FUNCTION_BLOCK FB_NormalWash IMPLEMENTS I_WashStrategy
VAR_INPUT
END_VAR
VAR_OUTPUT
END_VAR
VAR
END_VAR

{warning 'add method implementation '}
METHOD GetDuration
END_METHOD

{warning 'add method implementation '}
METHOD Start
END_METHOD

{warning 'add method implementation '}
METHOD Stop
END_METHOD

END_FUNCTION_BLOCK

(* stored: Version 1.1.0.1, ProductVersion 3.1.4024.16
   POU FB_NormalWash: Id {3a7130f4-98e7-4e05-a785-86970010f516}, SpecialFunc None
   Method GetDuration: Id {8a29e230-838d-43a3-91a5-5fe3abf18f33}
   Method Start: Id {5d96b91b-8f5c-464e-8848-f2528787bc71}
   Method Stop: Id {6de0414a-4a56-4f90-9038-d4f00b94516c} *)
